// SIMATIC S7-200 project (STEP 7-Micro/WIN), CPU 224 REL 01.12

ORGANIZATION_BLOCK PRINCIPAL:OB1
TITLE=COMENTARIOS DEL PROGRAMA
BEGIN
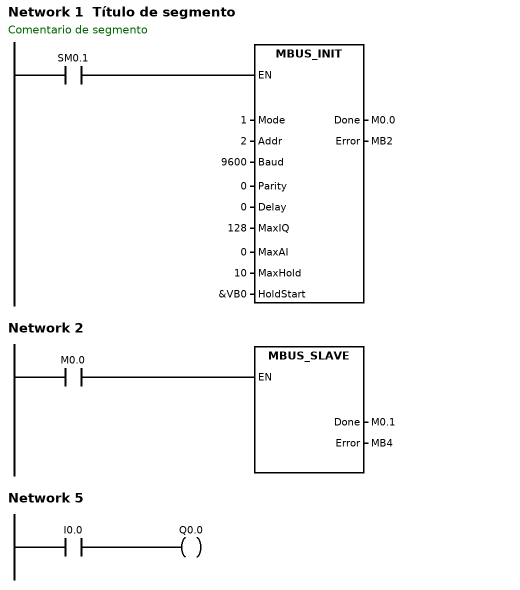
Network 1 // Título de segmento
// Comentario de segmento
LD     SM0.1
CALL   MBUS_INIT:SBR1, 1, 2, 9600, 0, 0, 128, 0, 10, &VB0, M0.0, MB2
Network 2
LD     M0.0
CALL   MBUS_SLAVE:SBR2, M0.1, MB4
Network 5
LD     I0.0
=      Q0.0
END_ORGANIZATION_BLOCK

// SBR1: protected block, not included

// SBR2: protected block, not included

// SBR3: protected block, not included
